(*
Der Soll-Tastgrad in Prozent gibt das Verhaeltnis der Sensorzustaende An zu Aus waehrend einer Aufnahme an.
*)
FUNCTION_BLOCK SignalDutyCycleRecorder
VAR_INPUT
  signal: BOOL;
END_VAR
VAR_OUTPUT
  recording_finished: BOOL;
  duty_cycle_ok: BOOL;
  error: BOOL;
END_VAR
VAR
  _record_delay: TIME := T#1S;
  _timeout: TIME := T#10S;
  _set_duty_cycle_in_percent: REAL := 90.0;
  signal_recorder: SignalTimeRecorder;
END_VAR

METHOD record
VAR_INPUT
  execute: BOOL;
END_VAR
VAR
  start_recording: BOOL;
END_VAR
VAR_INST
  t_timeout: TON;
  f_started_recording: F_TRIG;
  r_execute: R_TRIG;
END_VAR
r_execute(CLK:=execute);
IF r_execute.Q AND NOT error THEN
  recording_finished := FALSE;
  signal_recorder.record(execute:=FALSE);
  signal_recorder.reset();
END_IF

t_timeout(IN:=signal_recorder.started_recording, PT:=timeout);
IF t_timeout.Q THEN
  error := TRUE;
END_IF

start_recording := execute AND NOT error;

signal_recorder.record_delay := record_delay;
signal_recorder.signal := signal;
signal_recorder.record(execute:=start_recording);

f_started_recording(CLK:=signal_recorder.started_recording);
IF f_started_recording.Q THEN
  recording_finished := TRUE;
  duty_cycle_ok := signal_recorder.on_ratio * 100.0 >= set_duty_cycle_in_percent AND NOT error;
END_IF
END_METHOD

{attribute 'monitoring' := 'call'}
PROPERTY record_delay : TIME
GET
record_delay := _record_delay;
END_GET
SET
_record_delay := record_delay;
END_SET
END_PROPERTY

METHOD reset
VAR_INPUT
END_VAR
error := FALSE;
signal_recorder.reset();
END_METHOD

{attribute 'monitoring' := 'call'}
PROPERTY set_duty_cycle_in_percent : REAL
GET
set_duty_cycle_in_percent := _set_duty_cycle_in_percent;
END_GET
SET
VAR
  tastgrad: REAL;
END_VAR
IF set_duty_cycle_in_percent < 0 THEN
  tastgrad := 0.0;
ELSIF set_duty_cycle_in_percent > 100.0 THEN
  tastgrad := 100.0;
ELSE
  tastgrad := set_duty_cycle_in_percent;
END_IF
_set_duty_cycle_in_percent := tastgrad;
END_SET
END_PROPERTY

{attribute 'monitoring' := 'call'}
PROPERTY timeout : TIME
GET
timeout := _timeout;
END_GET
SET
_timeout := timeout;
END_SET
END_PROPERTY

END_FUNCTION_BLOCK

(* stored: Version 1.1.0.1, ProductVersion 3.1.4024.9
   POU SignalDutyCycleRecorder: Id {48bf5ea2-5b03-4893-b84f-88aefd604703}, SpecialFunc None
   Method record: Id {17d22e0b-d957-4eda-a6f5-290b7071cbb8}
   Property record_delay: Id {5171c9c4-9fcb-48f7-8e1e-b85a424f5f7f}
   Get Get: Id {1a34ded8-bb19-4757-b3a8-441ba08ef81a}
   Set Set: Id {bc1dc4c3-e9a3-4022-8730-c2215b3dfdd7}
   Method reset: Id {6cd35acf-0480-4475-b692-98cfceac7c54}
   Property set_duty_cycle_in_percent: Id {59a723f8-4e5d-4b58-99d8-75b48231e2af}
   Get Get: Id {72f77a1e-bd0d-41fd-a8e5-09584dc5aaaf}
   Set Set: Id {52f260b8-4373-4d3c-90c0-6759d6003d84}
   Property timeout: Id {20030a2c-9022-4d73-95a0-e81bf217fe2d}
   Get Get: Id {52fba5ed-1618-4f8f-8ca5-97eb2f417fea}
   Set Set: Id {74e8263c-a815-4593-9243-8ada5819ba9f} *)
